(* Logix 5000 project; controller SolisPLC_Vlad_CGL1 vendor 1 type 14 code 226 rev 36.11; software revision 36.00; part 3 of 3 *)
(* tags used below, declared in another part *)
   _AOI_Fah_to_Cel1 : _AOI_Fah_to_Cel;
   _AOI_Fah_to_Cel2 : _AOI_Fah_to_Cel;
   BoxID : DINT;
   BoxRejectSystem : DINT[100];
   BoxRejectSystem_CTRL : CONTROL;
   CasePackerBackUpTimer : TIMER;
   Conv1_Disch_BoxCounter : COUNTER;
   MC_Running : BOOL;
   MCO_T1 : TIMER;
   MCO_T10 : TIMER;
   MCO_T11 : TIMER;
   MCO_T2 : TIMER;
   MCO_T3 : TIMER;
   MCO_T4 : TIMER;
   MCO_T5 : TIMER;
   MCO_T6 : TIMER;
   MCO_T7 : TIMER;
   MCO_T8 : TIMER;
   MCO_T9 : TIMER;
   NarrowBox_CTU : COUNTER;
   PalletizerEMptyTimer : TIMER;
   PalletizerNeedsCase : BOOL;
   PartAssemblySeqStep : DINT;
   Placeholder1 : REAL;
   Placeholder2 : REAL;
   RejectID : DINT;
   S2_CasePackerBackedUp : BOOL;
   S2_Output : BOOL;
   S2_Output1 : BOOL;
   S2_Storage : BOOL;
   S2_Storage1 : BOOL;
   S2_SystemRunning : BOOL;
   SolisPLC_ONS : BOOL[64];
   TempC1 : REAL;
   TempC2 : REAL;
   TempC3 : REAL;
   TempF1 : REAL;
   TempF2 : REAL;
   TempF3 : REAL;
   WideBox_CTU : COUNTER;
   BOOL_IN_0 : BOOL;
   BOOL_IN_1 : BOOL;   // System Stop PB
   BOOL_OUT_0 : BOOL;   // STATUS - System Running
   BOOL_OUT_1 : BOOL;   // STATUS - System Stopped
   SolisPLC_B_IN_0 : BOOL;   // Start PB
   SolisPLC_B_IN_1 : BOOL;   // Stop PB
   SolisPLC_B_IN_10 : BOOL;   // System 2 - Palletizer Infeed Stop Sensor
   SolisPLC_B_IN_11 : BOOL;   // MC - Start PB
   SolisPLC_B_IN_12 : BOOL;   // MC - Stop PB
   SolisPLC_B_IN_15 : BOOL;   // MCO - Belt 2 Part Detected
   SolisPLC_B_IN_16 : BOOL;   // MCO - Belt 1 Part Detected
   SolisPLC_B_IN_2 : BOOL;   // Box Present Photo Eye [BLOCKED]
   SolisPLC_B_IN_3 : BOOL;   // Box Wide Photo Eye [BLOCKED]
   SolisPLC_B_IN_4 : BOOL;   // Pivot Arm Sensor
   SolisPLC_B_IN_6 : BOOL;   // System 2 - Start Push Button
   SolisPLC_B_IN_7 : BOOL;   // System 2 - Stop Push Button
   SolisPLC_B_IN_8 : BOOL;   // System 2 - Palletizer Infeed Sensor
   SolisPLC_B_IN_9 : BOOL;   // System 2 - Case Packer BackUp Sensor
   SolisPLC_B_OUT_0 : BOOL;   // Green Indicator
   SolisPLC_B_OUT_1 : BOOL;   // Red Indicator
   SolisPLC_B_OUT_10 : BOOL;   // MC - Discharge Conveyor RUN
   SolisPLC_B_OUT_11 : BOOL;   // MC - Robot Cell / CNC RUN
   SolisPLC_B_OUT_12 : BOOL;   // MC - Machining Center Produce Lids
   SolisPLC_B_OUT_13 : BOOL;
   SolisPLC_B_OUT_14 : BOOL;
   SolisPLC_B_OUT_15 : BOOL;
   SolisPLC_B_OUT_16 : BOOL;   // MCO - Belt 1 Clamp
   SolisPLC_B_OUT_17 : BOOL;   // MCO - Belt 2 Clamp
   SolisPLC_B_OUT_18 : BOOL;   // MCO - Pivot
   SolisPLC_B_OUT_19 : BOOL;   // MCO - Grabber
   SolisPLC_B_OUT_2 : BOOL;   // Belt Conveyor 1 Run
   SolisPLC_B_OUT_20 : BOOL;   // MCO - Place X Axis
   SolisPLC_B_OUT_21 : BOOL;   // MCO - Place Z Axis
   SolisPLC_B_OUT_22 : BOOL;   // MCO - Belt 2 Raise
   SolisPLC_B_OUT_3 : BOOL;   // Belt Conveyor 2 Run
   SolisPLC_B_OUT_4 : BOOL;   // Pivot Arm [TURN]
   SolisPLC_B_OUT_6 : BOOL;   // System 2 - Case Packer Enabled
   SolisPLC_B_OUT_7 : BOOL;   // System 2 - Case Packer Discharge Conveyor 1
   SolisPLC_B_OUT_8 : BOOL;   // System 2 - Palletizer Infeed Roller UP
   SolisPLC_B_OUT_9 : BOOL;   // MC - Infeed Conveyor RUN
   SolisPLC_F_OUT_0 : REAL;   // System 2 - Palletizer Infeed Prior to Stop Conveyor
   SolisPLC_F_OUT_1 : REAL;   // System 2 - Palletizer Infeed After Stop Conveyor
   SolisPLC_I_OUT_0 : INT;
   SolisPLC_I_OUT_1 : INT;   // Wide Box Counter
   SolisPLC_I_OUT_2 : INT;   // Narrow Box Counter
(* Tutorials, continued *)

ROUTINE _02_AOI   (* ladder *)
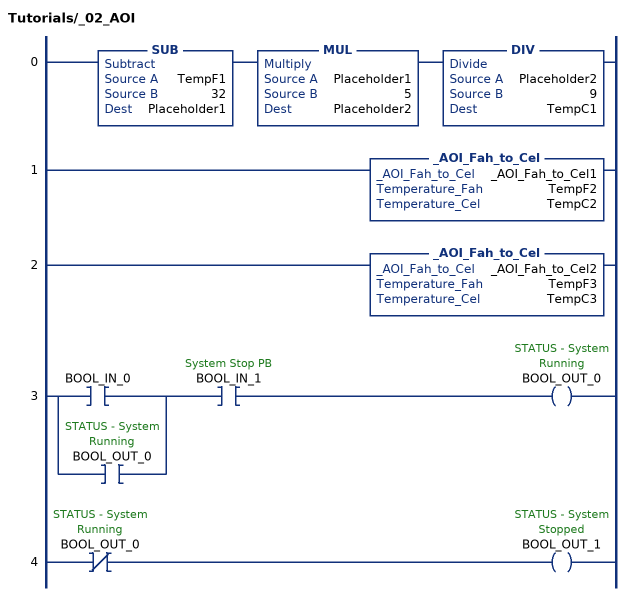
   0: SUB(TempF1,32,Placeholder1)MUL(Placeholder1,5,Placeholder2)DIV(Placeholder2,9,TempC1);
   1: _AOI_Fah_to_Cel(_AOI_Fah_to_Cel1,TempF2,TempC2);
   2: _AOI_Fah_to_Cel(_AOI_Fah_to_Cel2,TempF3,TempC3);
   3: [XIC(BOOL_IN_0) ,XIC(BOOL_OUT_0) ]XIC(BOOL_IN_1)OTE(BOOL_OUT_0);
   4: XIO(BOOL_OUT_0)OTE(BOOL_OUT_1);
END_ROUTINE

ROUTINE _03_FactoryIOSim   (* ladder *)
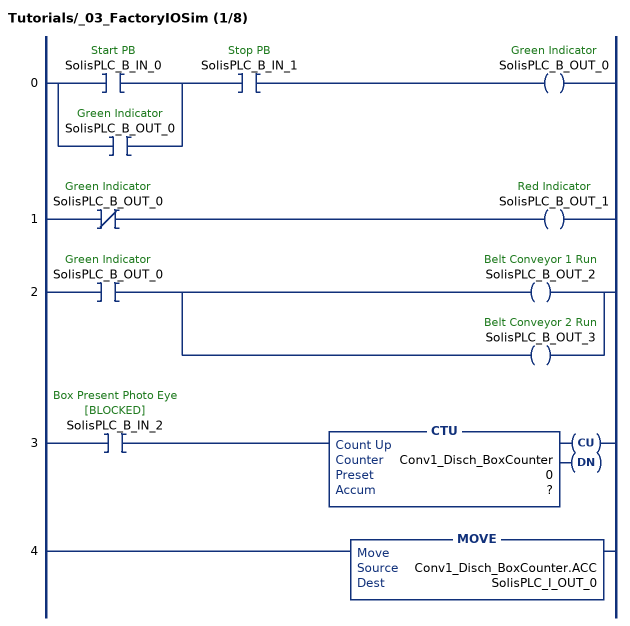
   0: [XIC(SolisPLC_B_IN_0) ,XIC(SolisPLC_B_OUT_0) ]XIC(SolisPLC_B_IN_1)OTE(SolisPLC_B_OUT_0);
   1: XIO(SolisPLC_B_OUT_0)OTE(SolisPLC_B_OUT_1);
   2: XIC(SolisPLC_B_OUT_0)[OTE(SolisPLC_B_OUT_2) ,OTE(SolisPLC_B_OUT_3) ];
   3: XIC(SolisPLC_B_IN_2)CTU(Conv1_Disch_BoxCounter,?,?);
   4: MOVE(Conv1_Disch_BoxCounter.ACC,SolisPLC_I_OUT_0);
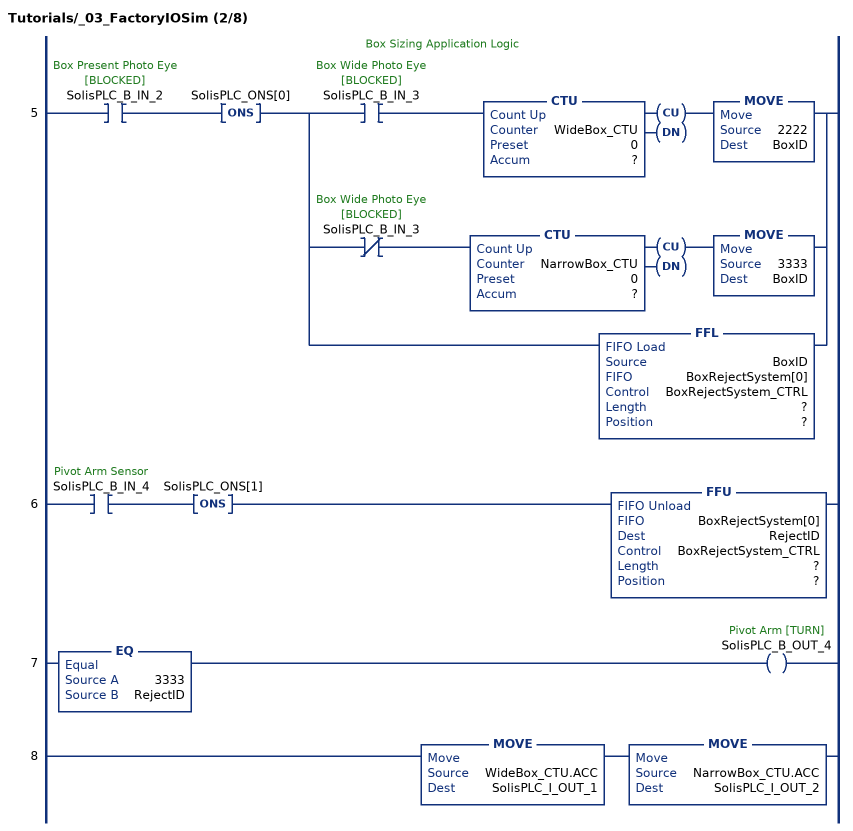
   // Box Sizing Application Logic
   5: XIC(SolisPLC_B_IN_2)ONS(SolisPLC_ONS[0])[XIC(SolisPLC_B_IN_3) CTU(WideBox_CTU,?,?) MOVE(2222,BoxID) ,XIO(SolisPLC_B_IN_3) CTU(NarrowBox_CTU,?,?) MOVE(3333,BoxID) ,FFL(BoxID,BoxRejectSystem[0],BoxRejectSystem_CTRL,?,?) ];
   6: XIC(SolisPLC_B_IN_4)ONS(SolisPLC_ONS[1])FFU(BoxRejectSystem[0],RejectID,BoxRejectSystem_CTRL,?,?);
   7: EQ(3333,RejectID)OTE(SolisPLC_B_OUT_4);
   8: MOVE(WideBox_CTU.ACC,SolisPLC_I_OUT_1)MOVE(NarrowBox_CTU.ACC,SolisPLC_I_OUT_2);
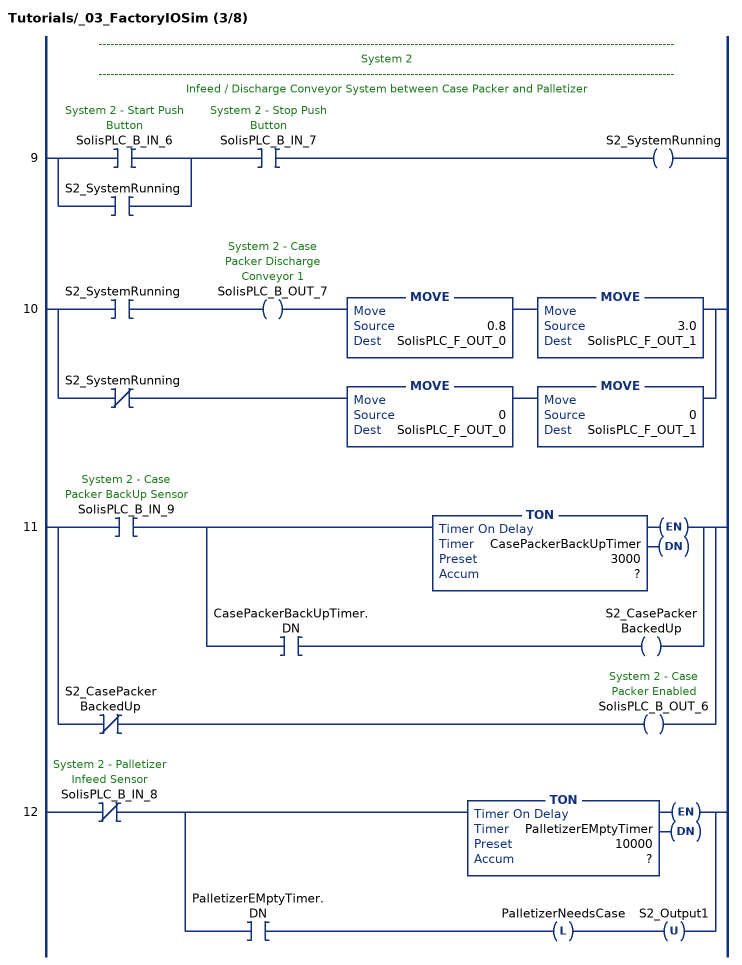
   // ------------------------------------------------------------------------------------------------------------------------------------------------
   // System 2
   // ------------------------------------------------------------------------------------------------------------------------------------------------
   // Infeed / Discharge Conveyor System between Case Packer and Palletizer
   9: [XIC(SolisPLC_B_IN_6) ,XIC(S2_SystemRunning) ]XIC(SolisPLC_B_IN_7)OTE(S2_SystemRunning);
   10: [XIC(S2_SystemRunning) OTE(SolisPLC_B_OUT_7) MOVE(0.8,SolisPLC_F_OUT_0) MOVE(3.0,SolisPLC_F_OUT_1) ,XIO(S2_SystemRunning) MOVE(0,SolisPLC_F_OUT_0) MOVE(0,SolisPLC_F_OUT_1) ];
   11: [XIC(SolisPLC_B_IN_9) [TON(CasePackerBackUpTimer,?,?) ,XIC(CasePackerBackUpTimer.DN) OTE(S2_CasePackerBackedUp) ] ,XIO(S2_CasePackerBackedUp) OTE(SolisPLC_B_OUT_6) ];
   12: XIO(SolisPLC_B_IN_8)[TON(PalletizerEMptyTimer,?,?) ,XIC(PalletizerEMptyTimer.DN) OTL(PalletizerNeedsCase) OTU(S2_Output1) ];
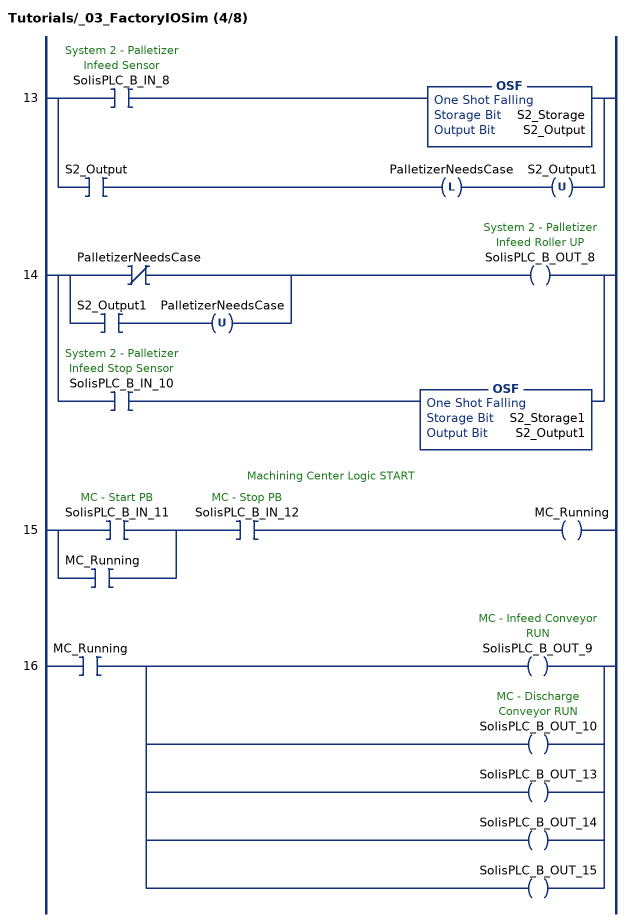
   13: [XIC(SolisPLC_B_IN_8) OSF(S2_Storage,S2_Output) ,XIC(S2_Output) OTL(PalletizerNeedsCase) OTU(S2_Output1) ];
   14: [[XIO(PalletizerNeedsCase) ,XIC(S2_Output1) OTU(PalletizerNeedsCase) ] OTE(SolisPLC_B_OUT_8) ,XIC(SolisPLC_B_IN_10) OSF(S2_Storage1,S2_Output1) ];
   // Machining Center Logic START
   15: [XIC(SolisPLC_B_IN_11) ,XIC(MC_Running) ]XIC(SolisPLC_B_IN_12)OTE(MC_Running);
   16: XIC(MC_Running)[OTE(SolisPLC_B_OUT_9) ,OTE(SolisPLC_B_OUT_10) ,OTE(SolisPLC_B_OUT_13) ,OTE(SolisPLC_B_OUT_14) ,OTE(SolisPLC_B_OUT_15) ];
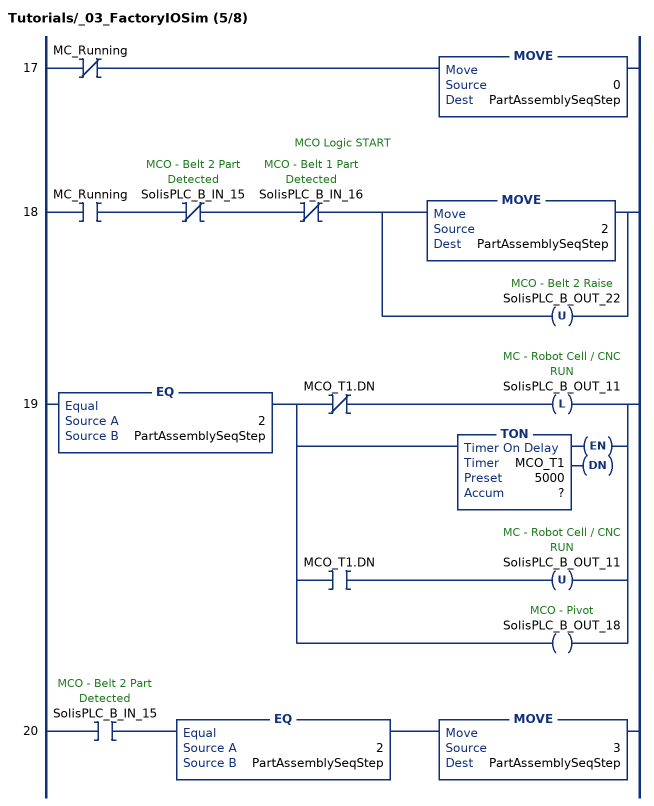
   17: XIO(MC_Running)MOVE(0,PartAssemblySeqStep);
   // MCO Logic START
   18: XIC(MC_Running)XIO(SolisPLC_B_IN_15)XIO(SolisPLC_B_IN_16)[MOVE(2,PartAssemblySeqStep) ,OTU(SolisPLC_B_OUT_22) ];
   19: EQ(2,PartAssemblySeqStep)[XIO(MCO_T1.DN) OTL(SolisPLC_B_OUT_11) ,TON(MCO_T1,?,?) ,XIC(MCO_T1.DN) OTU(SolisPLC_B_OUT_11) ,OTE(SolisPLC_B_OUT_18) ];
   20: XIC(SolisPLC_B_IN_15)EQ(2,PartAssemblySeqStep)MOVE(3,PartAssemblySeqStep);
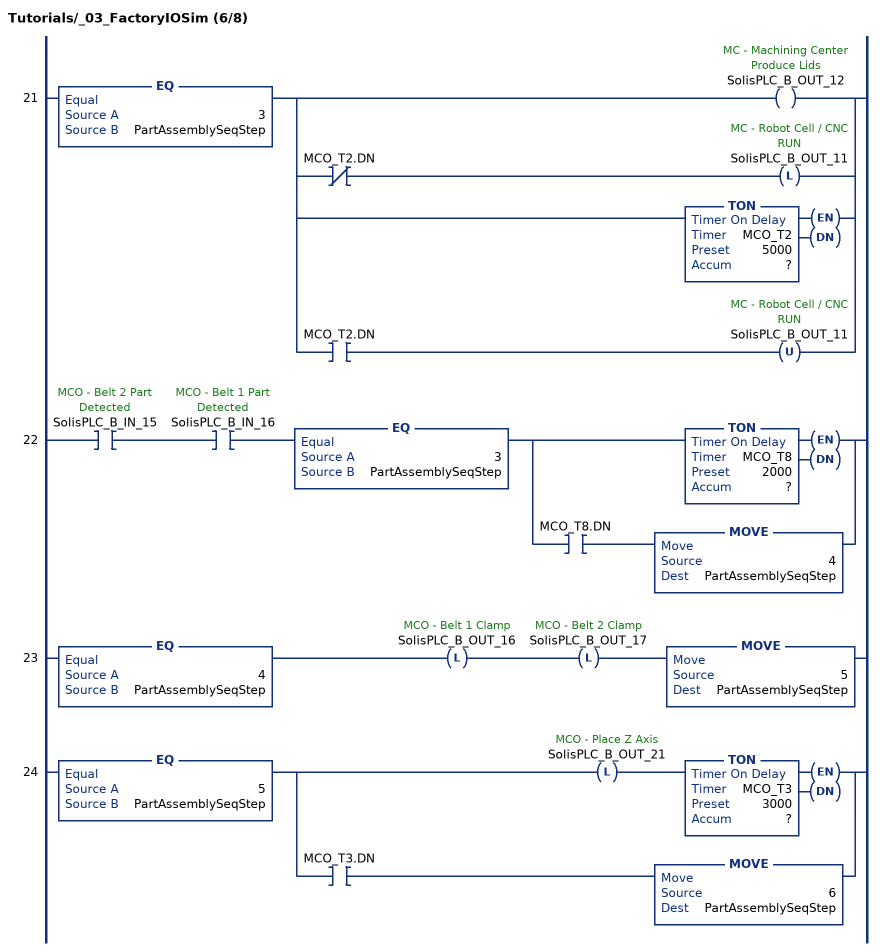
   21: EQ(3,PartAssemblySeqStep)[OTE(SolisPLC_B_OUT_12) ,XIO(MCO_T2.DN) OTL(SolisPLC_B_OUT_11) ,TON(MCO_T2,?,?) ,XIC(MCO_T2.DN) OTU(SolisPLC_B_OUT_11) ];
   22: XIC(SolisPLC_B_IN_15)XIC(SolisPLC_B_IN_16)EQ(3,PartAssemblySeqStep)[TON(MCO_T8,?,?) ,XIC(MCO_T8.DN) MOVE(4,PartAssemblySeqStep) ];
   23: EQ(4,PartAssemblySeqStep)OTL(SolisPLC_B_OUT_16)OTL(SolisPLC_B_OUT_17)MOVE(5,PartAssemblySeqStep);
   24: EQ(5,PartAssemblySeqStep)[OTL(SolisPLC_B_OUT_21) TON(MCO_T3,?,?) ,XIC(MCO_T3.DN) MOVE(6,PartAssemblySeqStep) ];
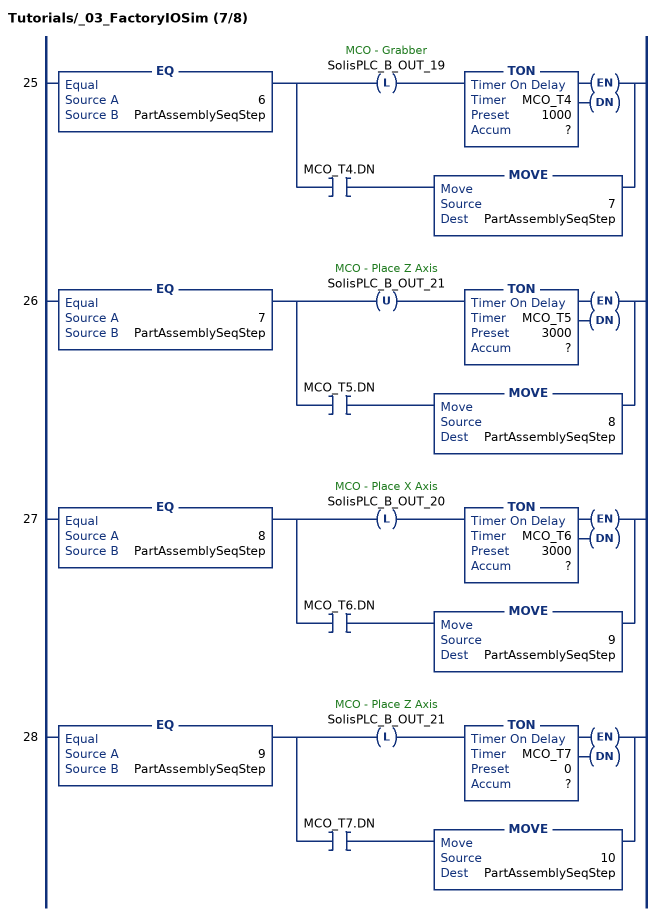
   25: EQ(6,PartAssemblySeqStep)[OTL(SolisPLC_B_OUT_19) TON(MCO_T4,?,?) ,XIC(MCO_T4.DN) MOVE(7,PartAssemblySeqStep) ];
   26: EQ(7,PartAssemblySeqStep)[OTU(SolisPLC_B_OUT_21) TON(MCO_T5,?,?) ,XIC(MCO_T5.DN) MOVE(8,PartAssemblySeqStep) ];
   27: EQ(8,PartAssemblySeqStep)[OTL(SolisPLC_B_OUT_20) TON(MCO_T6,?,?) ,XIC(MCO_T6.DN) MOVE(9,PartAssemblySeqStep) ];
   28: EQ(9,PartAssemblySeqStep)[OTL(SolisPLC_B_OUT_21) TON(MCO_T7,?,?) ,XIC(MCO_T7.DN) MOVE(10,PartAssemblySeqStep) ];
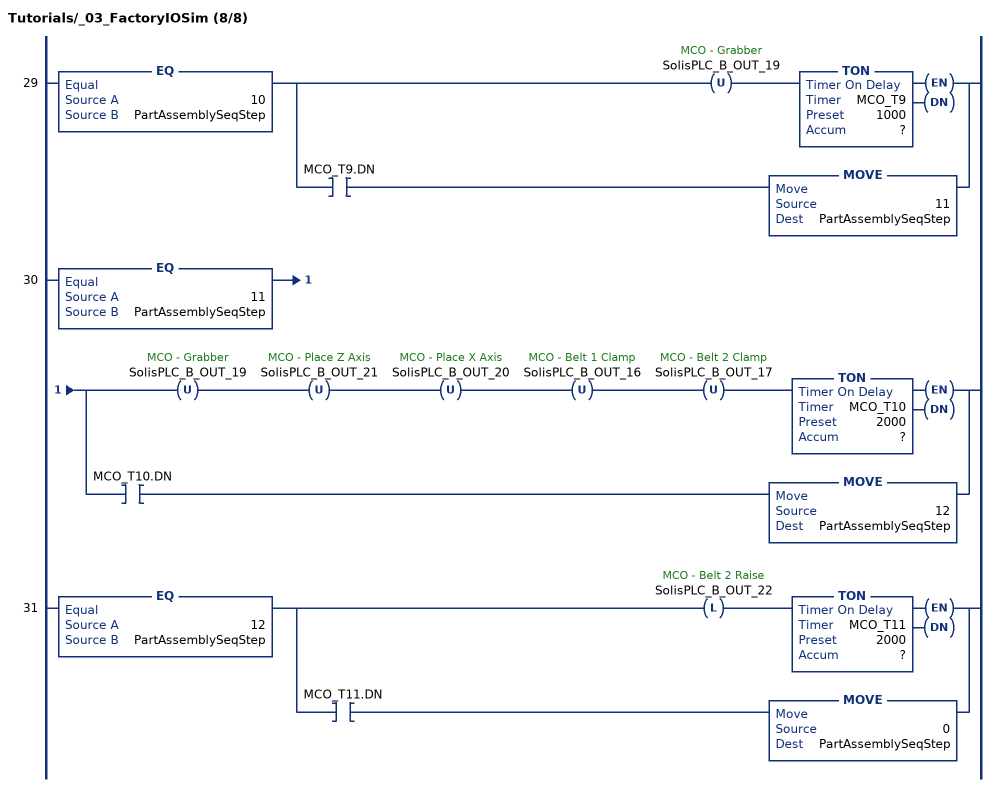
   29: EQ(10,PartAssemblySeqStep)[OTU(SolisPLC_B_OUT_19) TON(MCO_T9,?,?) ,XIC(MCO_T9.DN) MOVE(11,PartAssemblySeqStep) ];
   30: EQ(11,PartAssemblySeqStep)[OTU(SolisPLC_B_OUT_19) OTU(SolisPLC_B_OUT_21) OTU(SolisPLC_B_OUT_20) OTU(SolisPLC_B_OUT_16) OTU(SolisPLC_B_OUT_17) TON(MCO_T10,?,?) ,XIC(MCO_T10.DN) MOVE(12,PartAssemblySeqStep) ];
   31: EQ(12,PartAssemblySeqStep)[OTL(SolisPLC_B_OUT_22) TON(MCO_T11,?,?) ,XIC(MCO_T11.DN) MOVE(0,PartAssemblySeqStep) ];
END_ROUTINE
END_PROGRAM
